// TIA Portal project "cuacuonbyted" (V15)

(* hardware
DEVICE "S7-1200 station_2"  S7-1200 Station
   slot 0: "Rack_0"  S7-1200 Rack  Rack  V1.0
   slot 1: "PLC_2"  CPU 1212C DC/DC/DC  6ES7 212-1AE40-0XB0  V4.2
   slot 2: "DQ 8x24VDC _1"  SM 1222 DQ8 x 24VDC  6ES7 222-1BF32-0XB0  V2.0
   slot 3: "Battery board_1"  BB 1297 battery board  6ES7 297-0AX30-0XA0  V1.0
*)

// ===== PLC "PLC_2"  CPU 1212C DC/DC/DC =====

VAR_GLOBAL   // PLC tag table "Default tag table"
   "STOP" AT %M10.0 : Bool;
   "OPEN OUT(S1)" AT %M10.1 : Bool;
   "CLOSE OUT(S5)" AT %M10.2 : Bool;
   "OPEN IN(S2)" AT %M10.3 : Bool;
   "CLOSE IN(S4)" AT %M10.4 : Bool;
   "LIMIT UP(S3)" AT %M10.5 : Bool;
   "LIMIT DOWN(S6)" AT %M10.6 : Bool;
   "SAFE SENSOR(S7)" AT %M10.7 : Bool;
   "CLOSE DOOR DOWN" AT %Q0.0 : Bool;
   "OPEN DOOR UP" AT %Q0.1 : Bool;
   "WARNING LAMP" AT %Q0.2 : Bool;
   "Clock_Byte" AT %MB0 : Byte;
   "Clock_10Hz" AT %M0.0 : Bool;
   "Clock_5Hz" AT %M0.1 : Bool;
   "Clock_2.5Hz" AT %M0.2 : Bool;
   "Clock_2Hz" AT %M0.3 : Bool;
   "Clock_1.25Hz" AT %M0.4 : Bool;
   "Clock_1Hz" AT %M0.5 : Bool;
   "Clock_0.625Hz" AT %M0.6 : Bool;
   "Clock_0.5Hz" AT %M0.7 : Bool;
   "System_Byte" AT %MB1 : Byte;
   "FirstScan" AT %M1.0 : Bool;
   "DiagStatusUpdate" AT %M1.1 : Bool;
   "AlwaysTRUE" AT %M1.2 : Bool;
   "AlwaysFALSE" AT %M1.3 : Bool;
   "tagP" AT %M2.0 : Bool;
   "tagP1" AT %M2.1 : Bool;
   "tag11" AT %M2.3 : Bool;
END_VAR

// folder: System blocks/Program resources

DATA_BLOCK "IEC_Timer_0_DB_1"   // DB2
{ S7_Optimized_Access := 'TRUE' }
AUTHOR : Simatic
FAMILY : IEC
NAME : IEC_TMR
VERSION : 1.0
// stored: InstanceOfName IEC_TIMER
"IEC_TIMER"
BEGIN
END_DATA_BLOCK

// folder: (top level)

ORGANIZATION_BLOCK "Main"   // OB1, LAD, ProgramCycle
TITLE = "Main Program Sweep (Cycle)"
{ S7_Optimized_Access := 'TRUE' }
VERSION : 0.1
   VAR_TEMP   // added for the SCL form of the ladder/FBD networks
      _w1 : Bool;
      _w2 : Bool;
   END_VAR
BEGIN

REGION Network 1: Open the door
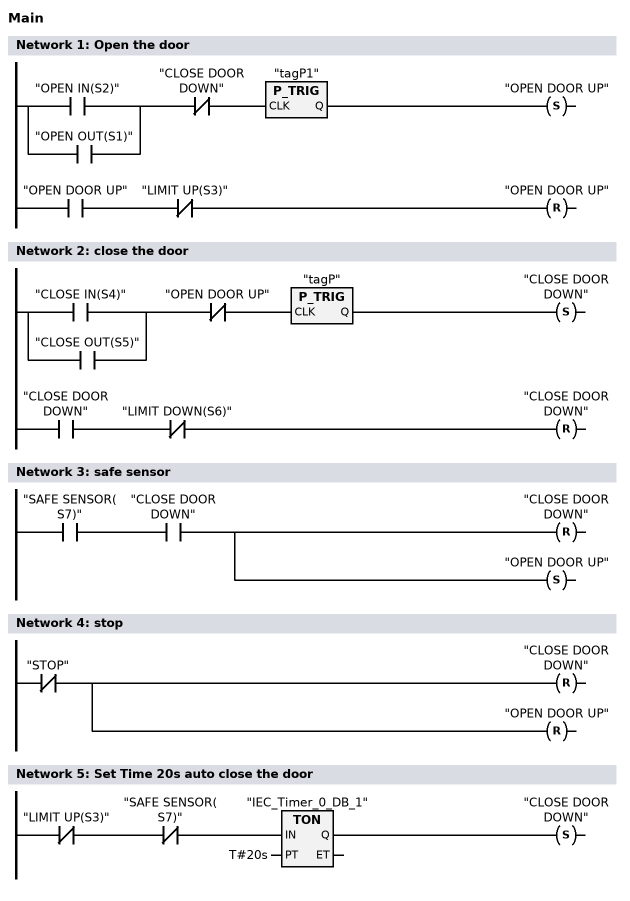
   RUNG wire#powerrail
      Contact( "OPEN IN(S2)" )
      wire#w1
      I_Contact( "CLOSE DOOR DOWN" )
      P_Trig( "tagP1" )
      S_Coil( "OPEN DOOR UP" )
   END_RUNG
   RUNG wire#powerrail
      Contact( "OPEN OUT(S1)" )
   END_RUNG wire#w1
   RUNG wire#powerrail
      Contact( "OPEN DOOR UP" )
      I_Contact( "LIMIT UP(S3)" )
      R_Coil( "OPEN DOOR UP" )
   END_RUNG
   // the same network as SCL:
   #_w1 := ("OPEN IN(S2)" OR "OPEN OUT(S1)") AND NOT "CLOSE DOOR DOWN";
   #_w2 := #_w1 AND NOT "tagP1";   // rising edge
   "tagP1" := #_w1;
   IF #_w2 THEN "OPEN DOOR UP" := TRUE; END_IF;
   IF "OPEN DOOR UP" AND NOT "LIMIT UP(S3)" THEN "OPEN DOOR UP" := FALSE; END_IF;
END_REGION

REGION Network 2: close the door
   RUNG wire#powerrail
      Contact( "CLOSE IN(S4)" )
      wire#w1
      I_Contact( "OPEN DOOR UP" )
      P_Trig( "tagP" )
      S_Coil( "CLOSE DOOR DOWN" )
   END_RUNG
   RUNG wire#powerrail
      Contact( "CLOSE OUT(S5)" )
   END_RUNG wire#w1
   RUNG wire#powerrail
      Contact( "CLOSE DOOR DOWN" )
      I_Contact( "LIMIT DOWN(S6)" )
      R_Coil( "CLOSE DOOR DOWN" )
   END_RUNG
   // the same network as SCL:
   #_w1 := ("CLOSE IN(S4)" OR "CLOSE OUT(S5)") AND NOT "OPEN DOOR UP";
   #_w2 := #_w1 AND NOT "tagP";   // rising edge
   "tagP" := #_w1;
   IF #_w2 THEN "CLOSE DOOR DOWN" := TRUE; END_IF;
   IF "CLOSE DOOR DOWN" AND NOT "LIMIT DOWN(S6)" THEN "CLOSE DOOR DOWN" := FALSE; END_IF;
END_REGION

REGION Network 3: safe sensor
   RUNG wire#powerrail
      Contact( "SAFE SENSOR(S7)" )
      Contact( "CLOSE DOOR DOWN" )
      wire#w1
      R_Coil( "CLOSE DOOR DOWN" )
   END_RUNG
   RUNG wire#w1
      S_Coil( "OPEN DOOR UP" )
   END_RUNG
   // the same network as SCL:
   #_w1 := "SAFE SENSOR(S7)" AND "CLOSE DOOR DOWN";
   IF #_w1 THEN
       "CLOSE DOOR DOWN" := FALSE;
       "OPEN DOOR UP" := TRUE;
   END_IF;
END_REGION

REGION Network 4: stop
   RUNG wire#powerrail
      I_Contact( "STOP" )
      wire#w1
      R_Coil( "CLOSE DOOR DOWN" )
   END_RUNG
   RUNG wire#w1
      R_Coil( "OPEN DOOR UP" )
   END_RUNG
   // the same network as SCL:
   IF NOT "STOP" THEN
       "CLOSE DOOR DOWN" := FALSE;
       "OPEN DOOR UP" := FALSE;
   END_IF;
END_REGION

REGION Network 5: Set Time 20s auto close the door
   "IEC_Timer_0_DB_1".TON(IN := NOT "LIMIT UP(S3)" AND NOT "SAFE SENSOR(S7)", PT := T#20s);
   IF "IEC_Timer_0_DB_1".Q THEN "CLOSE DOOR DOWN" := TRUE; END_IF;
END_REGION
END_ORGANIZATION_BLOCK